(*
SPDX-FileCopyrightText: © 2026 Oleksandr Tiutyk <trofimich@gmail.com>
SPDX-License-Identifier: MIT
License: https://opensource.org/license/mit
*)

{attribute 'qualified_only'}
{attribute 'strict'}
{attribute 'to_string'}
TYPE INTERSECTION_MODE :
(
	OFF,
	WORKING,
	FLASHING_YELLOW
);
END_TYPE

(* stored: Version 1.1.0.1
   DUT INTERSECTION_MODE: Id {b620d584-cfa1-4a4e-9931-6f98bba3c0d5} *)
